// TIA Portal V20 export
VAR_GLOBAL   // PLC tag table "IO_PLC_Centralizer_PLC_Functinal_Test_2"
   In_Functional_Test_Even AT %I300.0 : "IO_Device_Functinal_Test_Even";
   Out_Test_Parameters_Even AT %Q300.0 : "IO_Device_Test_Parameters_Even";
END_VAR
